// Mitsubishi GX Works2 project: Counter   PLC: Q03UDV

PROGRAM MAIN
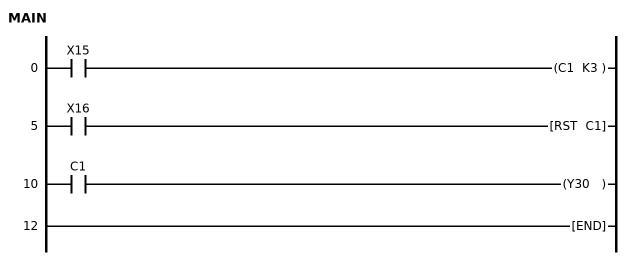
0     LD      X15
      OUT     C1 K3
5     LD      X16
      RST     C1
10    LD      C1
      OUT     Y30
12    END
END_PROGRAM
